// Mitsubishi GX Works2 project: FXPLC_Client_2   PLC: FX3U/FX3UC
// FXPLC_Client_2

PROGRAM MAIN
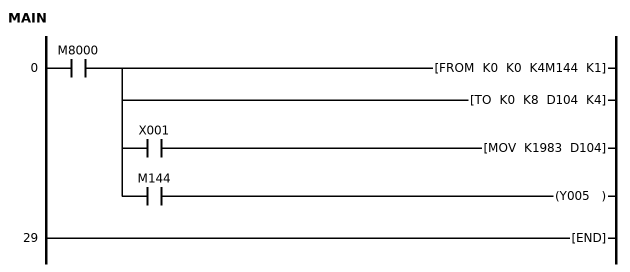
0     LD      M8000
      FROM    K0 K0 K4M144 K1
      TO      K0 K8 D104 K4
      MPS
      AND     X001
      MOV     K1983 D104
      MPP
      AND     M144
      OUT     Y005
29    END
END_PROGRAM
